VAR_GLOBAL CONSTANT
  MAX_PROCESS       : UINT := 3;
END_VAR
{attribute 'qualified_only'}
VAR_GLOBAL

  bDummy  : Bool;

END_VAR

(* stored: Version 1.1.0.1, ProductVersion 3.1.4024.13
   GVL GVL_APPLICATION: Id {b83de342-914f-4ad1-86ba-5efc40943708} *)
